// TIA Portal V19 export
VAR_GLOBAL   // PLC tag table "U3Em1_input"
   ngBeltForwardButton AT %I1.0 : Bool;
   ngBeltBackButton AT %I1.1 : Bool;
   materialDetectionU3Em1_6 AT %I220.5 : Bool;   // Material Detection 6
   materialDetectionU3Em1_8 AT %I220.7 : Bool;   // Material Detection 8
   materialDetectionU3Em1_7 AT %I220.6 : Bool;   // Material Detection 7
   materialDetectionU3Em1_4 AT %I220.3 : Bool;   // Material Detection 4
   materialDetectionU3Em1_2 AT %I220.1 : Bool;   // Material Detection 2
   materialDetectionU3Em1_5 AT %I220.4 : Bool;   // Material Detection 5
   materialDetectionU3Em1_1 AT %I220.0 : Bool;   // Material Detection 1
   materialDetectionU3Em1_3 AT %I220.2 : Bool;   // Material Detection 3
   materialDetectionU3Em1_9 AT %I221.0 : Bool;   // Material Detection 9
   ngStrapPositionDetectionU3Em1 AT %I221.1 : Bool;   // NG Pulling Belt Axis Motor Origin
END_VAR
